Staubli VAL3: calc_fuel.pgx

program calc_fuel(num x_nDiff, num& x_nFuel)
begin

  call util:range(0,x_nDiff+1,1,nRange)
  call math:sum(nRange, x_nFuel)

end
